TYPE E_VGC :
(

	Vented,
	AtVacuum,
	ERR_DiffPress,
	ERR_LostVac,
	ERR_ExtFault

);
END_TYPE

(* stored: Version 1.1.0.1, ProductVersion 3.1.4022.16
   DUT E_VGC: Id {fcf967d4-478c-4b51-acfa-c0d70935d131} *)
